// TIA Portal project "SortingLine_Project" (V18)

(* hardware
DEVICE "S7-1200 station_1"  S7-1200 Station
   slot 0: "Rack_0"  S7-1200 Rack  Rack  V1.0
   slot 1: "PLC_Sorting"  CPU 1214C DC/DC/DC  6ES7 214-1AG40-0XB0  V4.6
*)

// ===== PLC "PLC_Sorting"  CPU 1214C DC/DC/DC =====

VAR_GLOBAL   // PLC tag table "Factory_IO_Outputs"
   "Q_Counter" AT %QD30 : DInt;   // Digital totalizer display unit located on the operator panel.
   "Q_EntryConveyor" AT %Q0.1 : Bool;   // Drives the second section of the entry lane towards the turntable.
   "Q_FeederConveyor" AT %Q0.0 : Bool;   // Drives the first entry section right beneath the box emitter.
   "Q_GreenIndicator" AT %Q0.7 : Bool;   // Constant green indicates system is running active cycles.
   "Q_LeftConveyor" AT %Q0.5 : Bool;   // Drives the left clearance exit lane.
   "Q_Load" AT %Q0.2 : Bool;   // Runs internal turntable rollers forward to pull a box inside.
   "Q_RedIndicator" AT %Q1.1 : Bool;   // Constant red indicates system is idle/stopped.
   "Q_ResetLight" AT %Q1.3 : Bool;   // Active when safety is tripped and waiting for Reset.
   "Q_RightConveyor" AT %Q0.6 : Bool;   // Drives the right clearance exit lane.
   "Q_StartLight" AT %Q1.2 : Bool;   // Follows the Run state.
   "Q_StopLight" AT %Q1.4 : Bool;   // Active when cycle is offline.
   "Q_Turn" AT %Q0.4 : Bool;   // Swivels the turntable mechanism 90° clockwise.
   "Q_Unload" AT %Q0.3 : Bool;   // Runs internal turntable rollers backward to eject a box out to the left lane.
   "Q_YellowIndicator" AT %Q1.0 : Bool;   // Active on safety Fault or when system is in Manual mode.
   "Q_RemoverLeft" AT %Q1.5 : Bool;   // Instantly deletes boxes at the left exit limit.
   "Q_RemoverRight" AT %Q1.6 : Bool;   // Instantly deletes boxes at the right exit limit.
   "Q_Emit" AT %Q1.7 : Bool;   // Continuous TRUE spawns boxes sequentially.
END_VAR

VAR_GLOBAL   // PLC tag table "Factory_IO_Inputs"
   "I_atBack" AT %I2.1 : Bool;   // Confirms a box has fully cleared the entry area.
   "I_atEntry" AT %I0.0 : Bool;   // Detects box emergence.
   "I_atFront" AT %I0.6 : Bool;   // Prevents part collisions.
   "I_atLeftEntry" AT %I1.0 : Bool;   // Confirms the box has successfully transitioned onto the Left exit conveyor.
   "I_atLeftExit" AT %I1.2 : Bool;   // Drops to FALSE when a box reaches the left remover.
   "I_atLoadPosition" AT %I0.4 : Bool;   // TRUE when turntable is at 0° (aligned with entry).
   "I_atRightEntry" AT %I0.7 : Bool;   // Confirms the box has successfully transitioned onto the Right exit conveyor.
   "I_atRightExit" AT %I1.1 : Bool;   // Drops to FALSE when a box reaches the right remover.
   "I_atTurntableEntry" AT %I0.3 : Bool;   // Center reflective sensor inside the turntable. Used for precise stopping.
   "I_atUnloadPosition" AT %I0.5 : Bool;   // TRUE when turntable has completed its 90° clockwise rotation.
   "I_Auto" AT %I1.7 : Bool;   // Selector in Auto position.
   "I_Manual" AT %I2.2 : Bool;   // Selector in Manual position.
   "I_EmergencyStop" AT %I1.6 : Bool;   // TRUE when healthy, drops to FALSE when pressed.
   "I_LowBox" AT %I0.1 : Bool;   // Active (TRUE) for both low and high boxes.
   "I_Reset" AT %I1.4 : Bool;   // Clears safety fault latches.
   "I_Start" AT %I1.3 : Bool;   // Triggers the cycle run latch.
   "I_Stop" AT %I1.5 : Bool;   // TRUE at rest, drops to FALSE to request a cycle stop.
   "I_HighBox" AT %I0.2 : Bool;   // Active (TRUE) only alongside LowBox for high boxes.
END_VAR

TYPE "UDT_ActuatorCmd"
   STRUCT
      EntryConveyor : Bool;
      FeederConveyor : Bool;
      LeftConveyor : Bool;
      RightConveyor : Bool;
      Load : Bool;
      Unload : Bool;
      Turn : Bool;
      Emit : Bool;
      RemoverLeft : Bool := true;
      RemoverRight : Bool := true;
   END_STRUCT;
END_TYPE

DATA_BLOCK "DB_Machine"   // DB1
TITLE = Global Machine Status and Shared Data Registers
{ S7_Optimized_Access := 'TRUE' }
AUTHOR : HoraEmbedded
VERSION : 0.1
// Global Data Block (DB) serving as the main internal memory exchange registry for the system. Contains structured variables for system operating flags (Run, Fault, Modes), active part counters (Total, Left, Right), manual control parameters generated by the operator panel, and live engineering settings such as the box centering delay time variable.
   VAR
      Run : Bool;
      Fault : Bool;
      StopPending : Bool;
      AutoMode : Bool;
      ManualMode : Bool;
      CycleIdle : Bool;
      CountLeft : DInt;
      CountRight : DInt;
      CountTotal : DInt;
      AutoCmd : "UDT_ActuatorCmd";
      ManCmd : "UDT_ActuatorCmd";
      SortStep : DInt;
      ExitIdleHigh : Bool;
      ClearCounters : Bool;
      CenterTime : Time := T#2s;
   END_VAR
BEGIN
END_DATA_BLOCK

DATA_BLOCK "FB_ModeManager_DB"   // DB2
{ S7_Optimized_Access := 'TRUE' }
VERSION : 0.1
// stored: InstanceOfName FB_ModeManager
"FB_ModeManager"
BEGIN
END_DATA_BLOCK

DATA_BLOCK "FB_SortingLogic_DB"   // DB3
{ S7_Optimized_Access := 'TRUE' }
VERSION : 0.1
// stored: InstanceOfName FB_SortingLogic
"FB_SortingLogic"
BEGIN
END_DATA_BLOCK

FUNCTION_BLOCK "FB_ModeManager"   // FB1, LAD
TITLE = Machine Modes and Safety Interlocking Manager
{ S7_Optimized_Access := 'TRUE' }
AUTHOR : HoraEmbedded
VERSION : 0.1
// Monitors physical safety devices and panel inputs to manage operational states. Implements Normally Closed (NC) healthy monitoring for the Emergency Stop button, manages the manual safety fault latch (SR flip-flop), and handles the cycle stop requests (StopPending logic). It ensures a clean segregation between AutoMode and ManualMode to prevent overlapping operational commands.
   VAR_INPUT
      i_Start : Bool;   // Start pushbutton
      i_StopNC : Bool;   // Stop pushbutton
      i_EstopNC : Bool;   // Emergency stop
      i_Reset : Bool;   // Reset pushbutton
      i_Auto : Bool;   // Selector in Auto
      i_Manual : Bool;   // Selector in Manual
      i_CycleIdle : Bool;   // No box being processed
   END_VAR
   VAR_OUTPUT
      o_Run : Bool;
      o_Fault : Bool;
      o_StopPending : Bool;
      o_AutoMode : Bool;
      o_ManualMode : Bool;
   END_VAR
   VAR
      s_EdgeStart : Bool;   // Edge memory bits
      s_EdgeReset : Bool;   // Edge memory bits
   END_VAR
   VAR_TEMP
      t_StartPulse : Bool;   // One scan pulses
      t_ResetPulse : Bool;   // One scan pulses
   END_VAR
   VAR_TEMP   // added for the SCL form of the ladder/FBD networks
      _w1 : Bool;
   END_VAR
BEGIN

REGION Network 1: Auto mode
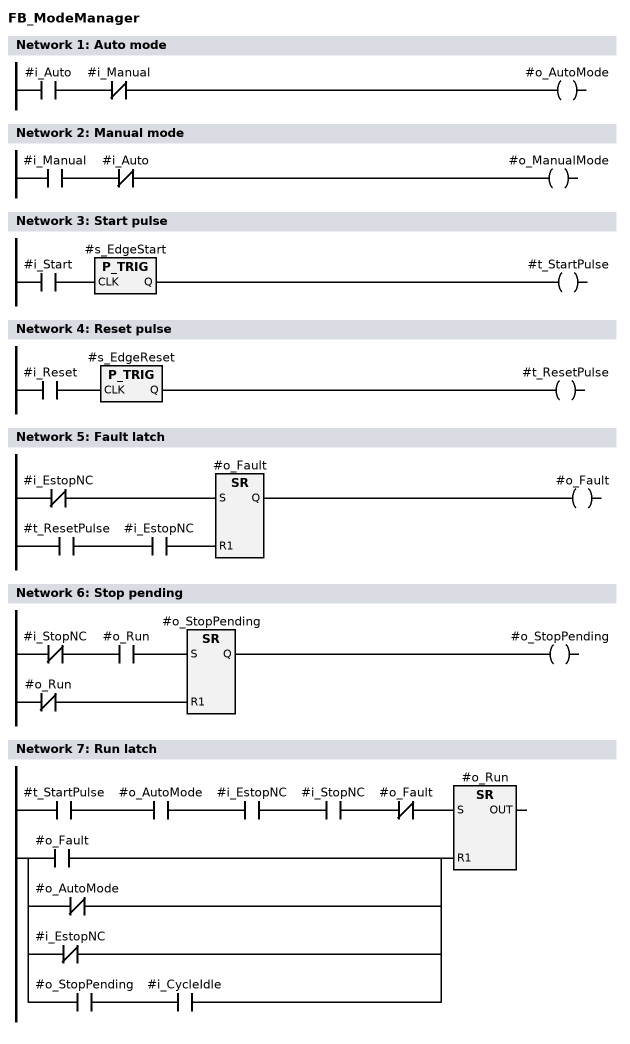
   RUNG wire#powerrail
      Contact( #i_Auto )
      I_Contact( #i_Manual )
      Coil( #o_AutoMode )
   END_RUNG
   // the same network as SCL:
   #o_AutoMode := #i_Auto AND NOT #i_Manual;
END_REGION

REGION Network 2: Manual mode
   RUNG wire#powerrail
      Contact( #i_Manual )
      I_Contact( #i_Auto )
      Coil( #o_ManualMode )
   END_RUNG
   // the same network as SCL:
   #o_ManualMode := #i_Manual AND NOT #i_Auto;
END_REGION

REGION Network 3: Start pulse
   RUNG wire#powerrail
      Contact( #i_Start )
      P_Trig( #s_EdgeStart )
      Coil( #t_StartPulse )
   END_RUNG
   // the same network as SCL:
   #_w1 := #i_Start AND NOT #s_EdgeStart;   // rising edge
   #s_EdgeStart := #i_Start;
   #t_StartPulse := #_w1;
END_REGION

REGION Network 4: Reset pulse
   RUNG wire#powerrail
      Contact( #i_Reset )
      P_Trig( #s_EdgeReset )
      Coil( #t_ResetPulse )
   END_RUNG
   // the same network as SCL:
   #_w1 := #i_Reset AND NOT #s_EdgeReset;   // rising edge
   #s_EdgeReset := #i_Reset;
   #t_ResetPulse := #_w1;
END_REGION

REGION Network 5: Fault latch
   RUNG wire#powerrail
      I_Contact( #i_EstopNC )
      S_SR(operand := #o_Fault, r1 := wire#w1)
      Coil( #o_Fault )
   END_RUNG
   RUNG wire#powerrail
      Contact( #t_ResetPulse )
      Contact( #i_EstopNC )
   END_RUNG wire#w1
   // the same network as SCL:
   IF NOT #i_EstopNC THEN
       #o_Fault := TRUE;   // SR flip-flop
   END_IF;
   IF #t_ResetPulse AND #i_EstopNC THEN #o_Fault := FALSE; END_IF;
   #o_Fault := #o_Fault;
END_REGION

REGION Network 6: Stop pending
   RUNG wire#powerrail
      I_Contact( #i_StopNC )
      Contact( #o_Run )
      S_SR(operand := #o_StopPending, r1 := wire#w1)
      Coil( #o_StopPending )
   END_RUNG
   RUNG wire#powerrail
      I_Contact( #o_Run )
   END_RUNG wire#w1
   // the same network as SCL:
   IF NOT #i_StopNC AND #o_Run THEN
       #o_StopPending := TRUE;   // SR flip-flop
   END_IF;
   IF NOT #o_Run THEN #o_StopPending := FALSE; END_IF;
   #o_StopPending := #o_StopPending;
END_REGION

REGION Network 7: Run latch
   RUNG wire#powerrail
      Contact( #t_StartPulse )
      Contact( #o_AutoMode )
      Contact( #i_EstopNC )
      Contact( #i_StopNC )
      I_Contact( #o_Fault )
      S_SR(operand := #o_Run, r1 := wire#w1)
   END_RUNG
   RUNG wire#powerrail
      Contact( #o_Fault )
   END_RUNG wire#w1
   RUNG wire#powerrail
      I_Contact( #o_AutoMode )
   END_RUNG wire#w1
   RUNG wire#powerrail
      I_Contact( #i_EstopNC )
   END_RUNG wire#w1
   RUNG wire#powerrail
      Contact( #o_StopPending )
      Contact( #i_CycleIdle )
   END_RUNG wire#w1
   // the same network as SCL:
   IF #t_StartPulse AND #o_AutoMode AND #i_EstopNC AND #i_StopNC AND NOT #o_Fault THEN
       #o_Run := TRUE;   // SR flip-flop
   END_IF;
   IF #o_Fault OR NOT #o_AutoMode OR NOT #i_EstopNC OR (#o_StopPending AND #i_CycleIdle) THEN
       #o_Run := FALSE;
   END_IF;
END_REGION
END_FUNCTION_BLOCK

FUNCTION_BLOCK "FB_SortingLogic"   // FB2, LAD
TITLE = Pipelined Box Sorting Sequence (State Machine)
{ S7_Optimized_Access := 'TRUE' }
AUTHOR : HoraEmbedded
VERSION : 0.1
// Implements the continuous automatic sorting sequence using a customized sequential state machine (Steps 0 to 5). Manages entry box generation, calculates sensor filtration via an independent centering timer block, tracks multiple parts in transit using dedicated software registers (In-Transit counters), and automatically routes boxes based on height measurements recorded by the light curtain.
   VAR_INPUT
      i_Run : Bool;
      i_StopPending : Bool;
      i_ClearCounters : Bool;
      i_ExitIdleHigh : Bool;
      i_atEntry : Bool;
      i_atLoadPosition : Bool;
      i_atTurntableEntry : Bool;
      i_atUnloadPosition : Bool;
      i_HighBox : Bool;
      i_atLeftEntry : Bool;
      i_atRightEntry : Bool;
      i_atLeftExit : Bool;
      i_atRightExit : Bool;
      i_CenterTime : Time;
      i_atFront : Bool;
   END_VAR
   VAR_OUTPUT
      o_CycleIdle : Bool;
      o_Step : DInt;
   END_VAR
   VAR_IN_OUT
      io_Cmd : "UDT_ActuatorCmd";
      io_CountLeft : DInt;
      io_CountRight : DInt;
      io_CountTotal : DInt;
   END_VAR
   VAR
      s_Step : DInt;
      s_SeenHigh : Bool;
      s_EdgeExitLeft : Bool;
      s_EdgeExitRight : Bool;
      s_TonEmit : IEC_TIMER;
      s_TonCenter : IEC_TIMER;
      s_atEntrySeen : Bool;
      s_LeftInTransit : DInt;
      s_RightInTransit : DInt;
      s_EdgeLeftEntry : Bool;
      s_EdgeRightEntry : Bool;
   END_VAR
   VAR_TEMP
      t_ExitLeftActive : Bool;
      t_ExitRightActive : Bool;
      t_ExitLeftPulse : Bool;
      t_ExitRightPulse : Bool;
      t_ChosenEntry : Bool;
      t_LeftEntryPulse : Bool;
      t_RightEntryPulse : Bool;
   END_VAR
   VAR_TEMP   // added for the SCL form of the ladder/FBD networks
      _w1 : Bool;
   END_VAR
BEGIN

REGION Network 1: exit left active
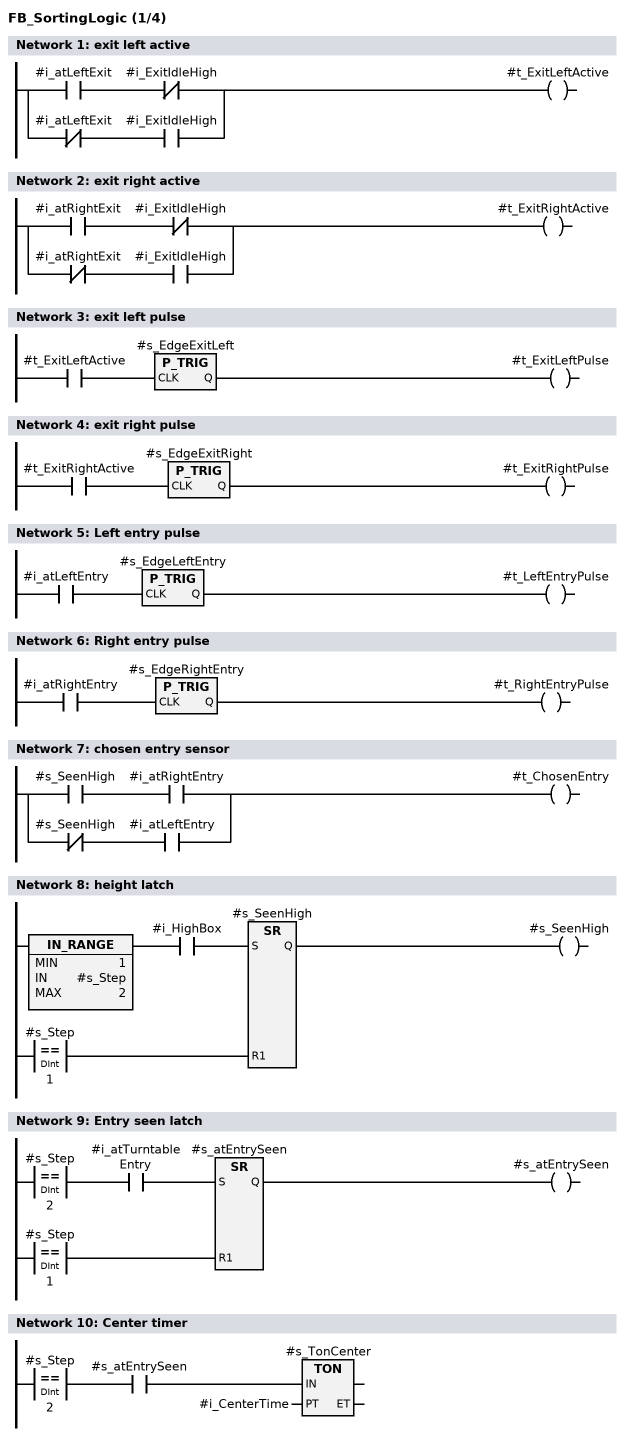
   RUNG wire#powerrail
      Contact( #i_atLeftExit )
      I_Contact( #i_ExitIdleHigh )
      wire#w1
      Coil( #t_ExitLeftActive )
   END_RUNG
   RUNG wire#powerrail
      I_Contact( #i_atLeftExit )
      Contact( #i_ExitIdleHigh )
   END_RUNG wire#w1
   // the same network as SCL:
   #t_ExitLeftActive := (#i_atLeftExit AND NOT #i_ExitIdleHigh) OR (NOT #i_atLeftExit AND #i_ExitIdleHigh);
END_REGION

REGION Network 2: exit right active
   RUNG wire#powerrail
      Contact( #i_atRightExit )
      I_Contact( #i_ExitIdleHigh )
      wire#w1
      Coil( #t_ExitRightActive )
   END_RUNG
   RUNG wire#powerrail
      I_Contact( #i_atRightExit )
      Contact( #i_ExitIdleHigh )
   END_RUNG wire#w1
   // the same network as SCL:
   #t_ExitRightActive := (#i_atRightExit AND NOT #i_ExitIdleHigh) OR (NOT #i_atRightExit AND #i_ExitIdleHigh);
END_REGION

REGION Network 3: exit left pulse
   RUNG wire#powerrail
      Contact( #t_ExitLeftActive )
      P_Trig( #s_EdgeExitLeft )
      Coil( #t_ExitLeftPulse )
   END_RUNG
   // the same network as SCL:
   #_w1 := #t_ExitLeftActive AND NOT #s_EdgeExitLeft;   // rising edge
   #s_EdgeExitLeft := #t_ExitLeftActive;
   #t_ExitLeftPulse := #_w1;
END_REGION

REGION Network 4: exit right pulse
   RUNG wire#powerrail
      Contact( #t_ExitRightActive )
      P_Trig( #s_EdgeExitRight )
      Coil( #t_ExitRightPulse )
   END_RUNG
   // the same network as SCL:
   #_w1 := #t_ExitRightActive AND NOT #s_EdgeExitRight;   // rising edge
   #s_EdgeExitRight := #t_ExitRightActive;
   #t_ExitRightPulse := #_w1;
END_REGION

REGION Network 5: Left entry pulse
   RUNG wire#powerrail
      Contact( #i_atLeftEntry )
      P_Trig( #s_EdgeLeftEntry )
      Coil( #t_LeftEntryPulse )
   END_RUNG
   // the same network as SCL:
   #_w1 := #i_atLeftEntry AND NOT #s_EdgeLeftEntry;   // rising edge
   #s_EdgeLeftEntry := #i_atLeftEntry;
   #t_LeftEntryPulse := #_w1;
END_REGION

REGION Network 6: Right entry pulse
   RUNG wire#powerrail
      Contact( #i_atRightEntry )
      P_Trig( #s_EdgeRightEntry )
      Coil( #t_RightEntryPulse )
   END_RUNG
   // the same network as SCL:
   #_w1 := #i_atRightEntry AND NOT #s_EdgeRightEntry;   // rising edge
   #s_EdgeRightEntry := #i_atRightEntry;
   #t_RightEntryPulse := #_w1;
END_REGION

REGION Network 7: chosen entry sensor
   RUNG wire#powerrail
      Contact( #s_SeenHigh )
      Contact( #i_atRightEntry )
      wire#w1
      Coil( #t_ChosenEntry )
   END_RUNG
   RUNG wire#powerrail
      I_Contact( #s_SeenHigh )
      Contact( #i_atLeftEntry )
   END_RUNG wire#w1
   // the same network as SCL:
   #t_ChosenEntry := (#s_SeenHigh AND #i_atRightEntry) OR (NOT #s_SeenHigh AND #i_atLeftEntry);
END_REGION

REGION Network 8: height latch
   RUNG wire#powerrail
      { S7_Templates := "SrcType := DInt" } InRange(min := 1, in := #s_Step, max := 2)
      Contact( #i_HighBox )
      S_SR(operand := #s_SeenHigh, r1 := wire#w1)
      Coil( #s_SeenHigh )
   END_RUNG
   RUNG wire#powerrail
      { S7_Templates := "SrcType := DInt" } EQ_Contact(in1 := #s_Step, in2 := 1)
   END_RUNG wire#w1
   // the same network as SCL:
   IF (1 <= #s_Step) AND (#s_Step <= 2) AND #i_HighBox THEN
       #s_SeenHigh := TRUE;   // SR flip-flop
   END_IF;
   IF #s_Step = 1 THEN #s_SeenHigh := FALSE; END_IF;
   #s_SeenHigh := #s_SeenHigh;
END_REGION

REGION Network 9: Entry seen latch
   RUNG wire#powerrail
      { S7_Templates := "SrcType := DInt" } EQ_Contact(in1 := #s_Step, in2 := 2)
      Contact( #i_atTurntableEntry )
      S_SR(operand := #s_atEntrySeen, r1 := wire#w1)
      Coil( #s_atEntrySeen )
   END_RUNG
   RUNG wire#powerrail
      { S7_Templates := "SrcType := DInt" } EQ_Contact(in1 := #s_Step, in2 := 1)
   END_RUNG wire#w1
   // the same network as SCL:
   IF (#s_Step = 2) AND #i_atTurntableEntry THEN
       #s_atEntrySeen := TRUE;   // SR flip-flop
   END_IF;
   IF #s_Step = 1 THEN #s_atEntrySeen := FALSE; END_IF;
   #s_atEntrySeen := #s_atEntrySeen;
END_REGION

REGION Network 10: Center timer
   #s_TonCenter.TON(IN := (#s_Step = 2) AND #s_atEntrySeen, PT := #i_CenterTime);
END_REGION

REGION Network 11: T4 to 5 (#s_Step := 5)
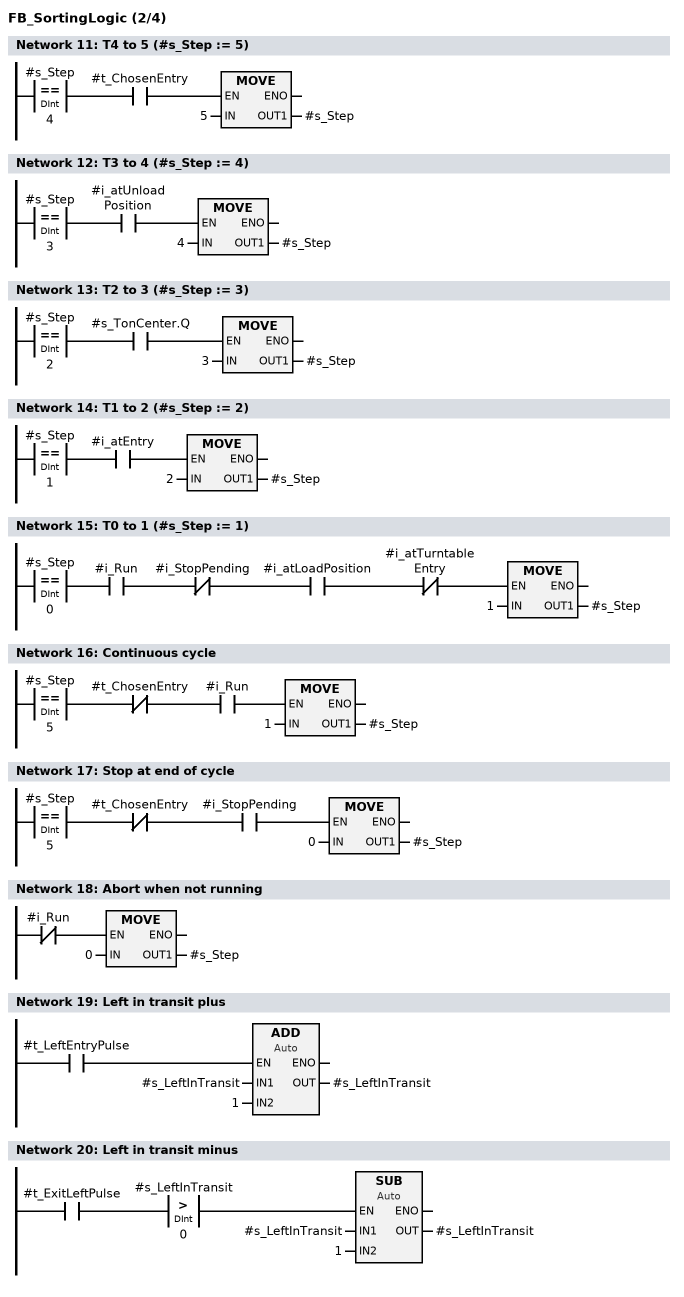
   RUNG wire#powerrail
      { S7_Templates := "SrcType := DInt" } EQ_Contact(in1 := #s_Step, in2 := 4)
      Contact( #t_ChosenEntry )
      Move(in := 5, out1 => #s_Step)
   END_RUNG
   // the same network as SCL:
   IF (#s_Step = 4) AND #t_ChosenEntry THEN #s_Step := 5; END_IF;
END_REGION

REGION Network 12: T3 to 4 (#s_Step := 4)
   RUNG wire#powerrail
      { S7_Templates := "SrcType := DInt" } EQ_Contact(in1 := #s_Step, in2 := 3)
      Contact( #i_atUnloadPosition )
      Move(in := 4, out1 => #s_Step)
   END_RUNG
   // the same network as SCL:
   IF (#s_Step = 3) AND #i_atUnloadPosition THEN #s_Step := 4; END_IF;
END_REGION

REGION Network 13: T2 to 3 (#s_Step := 3)
   RUNG wire#powerrail
      { S7_Templates := "SrcType := DInt" } EQ_Contact(in1 := #s_Step, in2 := 2)
      Contact( #s_TonCenter.Q )
      Move(in := 3, out1 => #s_Step)
   END_RUNG
   // the same network as SCL:
   IF (#s_Step = 2) AND #s_TonCenter.Q THEN #s_Step := 3; END_IF;
END_REGION

REGION Network 14: T1 to 2 (#s_Step := 2)
   RUNG wire#powerrail
      { S7_Templates := "SrcType := DInt" } EQ_Contact(in1 := #s_Step, in2 := 1)
      Contact( #i_atEntry )
      Move(in := 2, out1 => #s_Step)
   END_RUNG
   // the same network as SCL:
   IF (#s_Step = 1) AND #i_atEntry THEN #s_Step := 2; END_IF;
END_REGION

REGION Network 15: T0 to 1 (#s_Step := 1)
   RUNG wire#powerrail
      { S7_Templates := "SrcType := DInt" } EQ_Contact(in1 := #s_Step, in2 := 0)
      Contact( #i_Run )
      I_Contact( #i_StopPending )
      Contact( #i_atLoadPosition )
      I_Contact( #i_atTurntableEntry )
      Move(in := 1, out1 => #s_Step)
   END_RUNG
   // the same network as SCL:
   IF (#s_Step = 0) AND #i_Run AND NOT #i_StopPending AND #i_atLoadPosition AND NOT #i_atTurntableEntry THEN
       #s_Step := 1;
   END_IF;
END_REGION

REGION Network 16: Continuous cycle
   RUNG wire#powerrail
      { S7_Templates := "SrcType := DInt" } EQ_Contact(in1 := #s_Step, in2 := 5)
      I_Contact( #t_ChosenEntry )
      Contact( #i_Run )
      Move(in := 1, out1 => #s_Step)
   END_RUNG
   // the same network as SCL:
   IF (#s_Step = 5) AND NOT #t_ChosenEntry AND #i_Run THEN #s_Step := 1; END_IF;
END_REGION

REGION Network 17: Stop at end of cycle
   RUNG wire#powerrail
      { S7_Templates := "SrcType := DInt" } EQ_Contact(in1 := #s_Step, in2 := 5)
      I_Contact( #t_ChosenEntry )
      Contact( #i_StopPending )
      Move(in := 0, out1 => #s_Step)
   END_RUNG
   // the same network as SCL:
   IF (#s_Step = 5) AND NOT #t_ChosenEntry AND #i_StopPending THEN #s_Step := 0; END_IF;
END_REGION

REGION Network 18: Abort when not running
   RUNG wire#powerrail
      I_Contact( #i_Run )
      Move(in := 0, out1 => #s_Step)
   END_RUNG
   // the same network as SCL:
   IF NOT #i_Run THEN #s_Step := 0; END_IF;
END_REGION

REGION Network 19: Left in transit plus
   RUNG wire#powerrail
      Contact( #t_LeftEntryPulse )
      Add(in1 := #s_LeftInTransit, in2 := 1, out => #s_LeftInTransit)
   END_RUNG
   // the same network as SCL:
   IF #t_LeftEntryPulse THEN #s_LeftInTransit := #s_LeftInTransit + 1; END_IF;
END_REGION

REGION Network 20: Left in transit minus
   RUNG wire#powerrail
      Contact( #t_ExitLeftPulse )
      { S7_Templates := "SrcType := DInt" } GT_Contact(in1 := #s_LeftInTransit, in2 := 0)
      Sub(in1 := #s_LeftInTransit, in2 := 1, out => #s_LeftInTransit)
   END_RUNG
   // the same network as SCL:
   IF #t_ExitLeftPulse AND (#s_LeftInTransit > 0) THEN #s_LeftInTransit := #s_LeftInTransit - 1; END_IF;
END_REGION

REGION Network 21: Left in transit clear
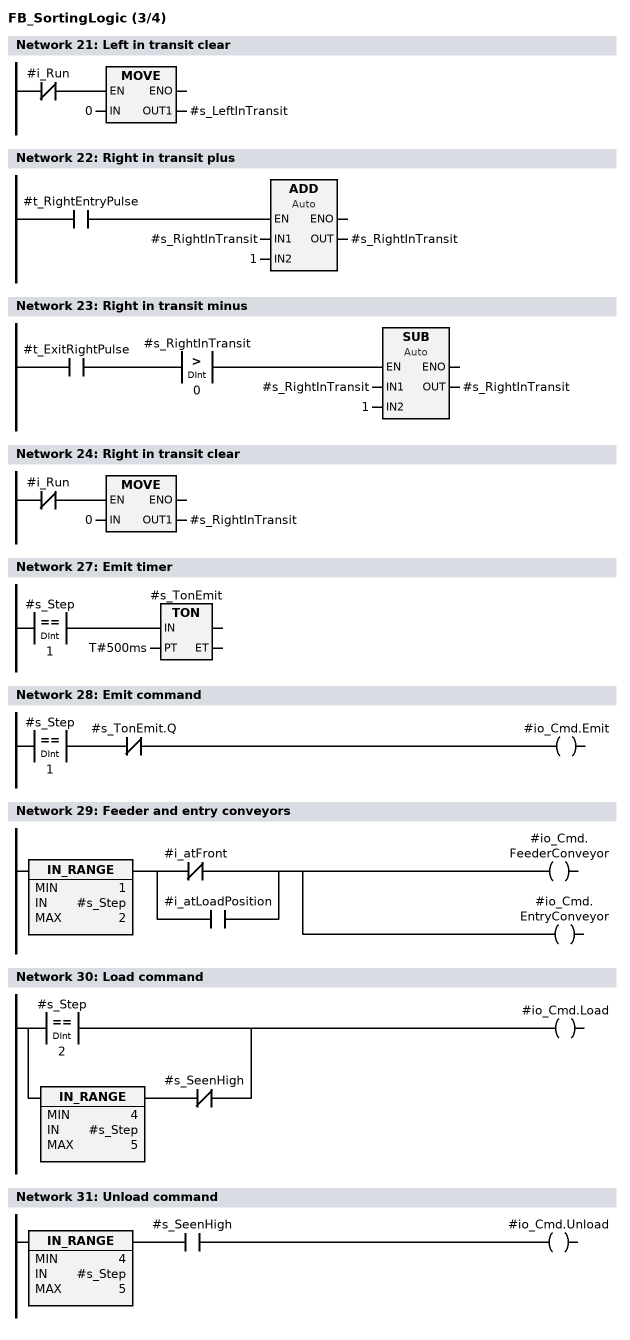
   RUNG wire#powerrail
      I_Contact( #i_Run )
      Move(in := 0, out1 => #s_LeftInTransit)
   END_RUNG
   // the same network as SCL:
   IF NOT #i_Run THEN #s_LeftInTransit := 0; END_IF;
END_REGION

REGION Network 22: Right in transit plus
   RUNG wire#powerrail
      Contact( #t_RightEntryPulse )
      Add(in1 := #s_RightInTransit, in2 := 1, out => #s_RightInTransit)
   END_RUNG
   // the same network as SCL:
   IF #t_RightEntryPulse THEN #s_RightInTransit := #s_RightInTransit + 1; END_IF;
END_REGION

REGION Network 23: Right in transit minus
   RUNG wire#powerrail
      Contact( #t_ExitRightPulse )
      { S7_Templates := "SrcType := DInt" } GT_Contact(in1 := #s_RightInTransit, in2 := 0)
      Sub(in1 := #s_RightInTransit, in2 := 1, out => #s_RightInTransit)
   END_RUNG
   // the same network as SCL:
   IF #t_ExitRightPulse AND (#s_RightInTransit > 0) THEN #s_RightInTransit := #s_RightInTransit - 1; END_IF;
END_REGION

REGION Network 24: Right in transit clear
   RUNG wire#powerrail
      I_Contact( #i_Run )
      Move(in := 0, out1 => #s_RightInTransit)
   END_RUNG
   // the same network as SCL:
   IF NOT #i_Run THEN #s_RightInTransit := 0; END_IF;
END_REGION

REGION Network 25: Continuous cycle
END_REGION

REGION Network 26: Stop at end of cycle
END_REGION

REGION Network 27: Emit timer
   #s_TonEmit.TON(IN := #s_Step = 1, PT := T#500ms);
END_REGION

REGION Network 28: Emit command
   RUNG wire#powerrail
      { S7_Templates := "SrcType := DInt" } EQ_Contact(in1 := #s_Step, in2 := 1)
      I_Contact( #s_TonEmit.Q )
      Coil( #io_Cmd.Emit )
   END_RUNG
   // the same network as SCL:
   #io_Cmd.Emit := (#s_Step = 1) AND NOT #s_TonEmit.Q;
END_REGION

REGION Network 29: Feeder and entry conveyors
   RUNG wire#powerrail
      { S7_Templates := "SrcType := DInt" } InRange(min := 1, in := #s_Step, max := 2)
      wire#w1
      I_Contact( #i_atFront )
      wire#w2
      Coil( #io_Cmd.FeederConveyor )
   END_RUNG
   RUNG wire#w1
      Contact( #i_atLoadPosition )
   END_RUNG wire#w2
   RUNG wire#w2
      Coil( #io_Cmd.EntryConveyor )
   END_RUNG
   // the same network as SCL:
   #io_Cmd.FeederConveyor := (1 <= #s_Step) AND (#s_Step <= 2) AND (NOT #i_atFront OR #i_atLoadPosition);
   #io_Cmd.EntryConveyor := #io_Cmd.FeederConveyor;
END_REGION

REGION Network 30: Load command
   RUNG wire#powerrail
      { S7_Templates := "SrcType := DInt" } EQ_Contact(in1 := #s_Step, in2 := 2)
      wire#w1
      Coil( #io_Cmd.Load )
   END_RUNG
   RUNG wire#powerrail
      { S7_Templates := "SrcType := DInt" } InRange(min := 4, in := #s_Step, max := 5)
      I_Contact( #s_SeenHigh )
   END_RUNG wire#w1
   // the same network as SCL:
   #io_Cmd.Load := (#s_Step = 2) OR ((4 <= #s_Step) AND (#s_Step <= 5) AND NOT #s_SeenHigh);
END_REGION

REGION Network 31: Unload command
   RUNG wire#powerrail
      { S7_Templates := "SrcType := DInt" } InRange(min := 4, in := #s_Step, max := 5)
      Contact( #s_SeenHigh )
      Coil( #io_Cmd.Unload )
   END_RUNG
   // the same network as SCL:
   #io_Cmd.Unload := (4 <= #s_Step) AND (#s_Step <= 5) AND #s_SeenHigh;
END_REGION

REGION Network 32: Turn command
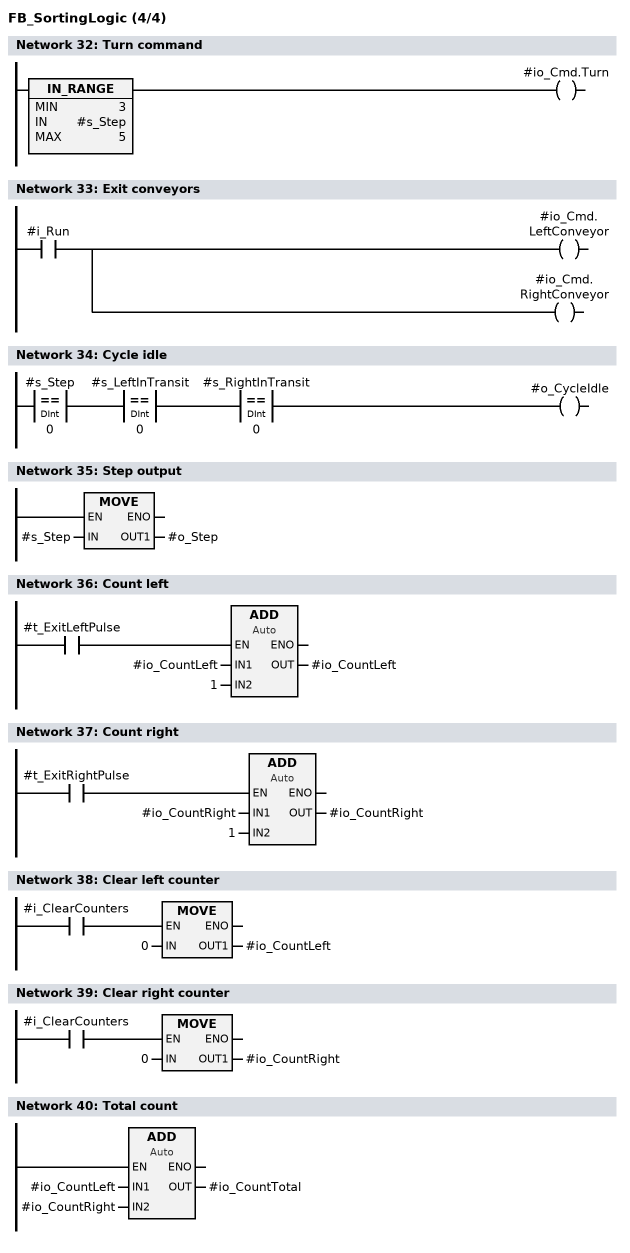
   RUNG wire#powerrail
      { S7_Templates := "SrcType := DInt" } InRange(min := 3, in := #s_Step, max := 5)
      Coil( #io_Cmd.Turn )
   END_RUNG
   // the same network as SCL:
   #io_Cmd.Turn := (3 <= #s_Step) AND (#s_Step <= 5);
END_REGION

REGION Network 33: Exit conveyors
   RUNG wire#powerrail
      Contact( #i_Run )
      wire#w1
      Coil( #io_Cmd.LeftConveyor )
   END_RUNG
   RUNG wire#w1
      Coil( #io_Cmd.RightConveyor )
   END_RUNG
   // the same network as SCL:
   #io_Cmd.LeftConveyor := #i_Run;
   #io_Cmd.RightConveyor := #i_Run;
END_REGION

REGION Network 34: Cycle idle
   RUNG wire#powerrail
      { S7_Templates := "SrcType := DInt" } EQ_Contact(in1 := #s_Step, in2 := 0)
      { S7_Templates := "SrcType := DInt" } EQ_Contact(in1 := #s_LeftInTransit, in2 := 0)
      { S7_Templates := "SrcType := DInt" } EQ_Contact(in1 := #s_RightInTransit, in2 := 0)
      Coil( #o_CycleIdle )
   END_RUNG
   // the same network as SCL:
   #o_CycleIdle := (#s_Step = 0) AND (#s_LeftInTransit = 0) AND (#s_RightInTransit = 0);
END_REGION

REGION Network 35: Step output
   RUNG wire#powerrail
      Move(in := #s_Step, out1 => #o_Step)
   END_RUNG
   // the same network as SCL:
   #o_Step := #s_Step;
END_REGION

REGION Network 36: Count left
   RUNG wire#powerrail
      Contact( #t_ExitLeftPulse )
      Add(in1 := #io_CountLeft, in2 := 1, out => #io_CountLeft)
   END_RUNG
   // the same network as SCL:
   IF #t_ExitLeftPulse THEN #io_CountLeft := #io_CountLeft + 1; END_IF;
END_REGION

REGION Network 37: Count right
   RUNG wire#powerrail
      Contact( #t_ExitRightPulse )
      Add(in1 := #io_CountRight, in2 := 1, out => #io_CountRight)
   END_RUNG
   // the same network as SCL:
   IF #t_ExitRightPulse THEN #io_CountRight := #io_CountRight + 1; END_IF;
END_REGION

REGION Network 38: Clear left counter
   RUNG wire#powerrail
      Contact( #i_ClearCounters )
      Move(in := 0, out1 => #io_CountLeft)
   END_RUNG
   // the same network as SCL:
   IF #i_ClearCounters THEN #io_CountLeft := 0; END_IF;
END_REGION

REGION Network 39: Clear right counter
   RUNG wire#powerrail
      Contact( #i_ClearCounters )
      Move(in := 0, out1 => #io_CountRight)
   END_RUNG
   // the same network as SCL:
   IF #i_ClearCounters THEN #io_CountRight := 0; END_IF;
END_REGION

REGION Network 40: Total count
   RUNG wire#powerrail
      Add(in1 := #io_CountLeft, in2 := #io_CountRight, out => #io_CountTotal)
   END_RUNG
   // the same network as SCL:
   #io_CountTotal := #io_CountLeft + #io_CountRight;
END_REGION
END_FUNCTION_BLOCK

FUNCTION "FC_outputs" : Void   // FC1, LAD
TITLE = Centralized Output Gating and Hardware Interlocks
{ S7_Optimized_Access := 'TRUE' }
AUTHOR : HoraEmbedded
VERSION : 0.1
// Serves as the single source of truth for all physical digital and analog outputs directed to the Factory I/O simulation panel. It gathers automatic commands generated by the state machine and manual commands from the watch table. It applies strict hardware safety interlocks (System Enable bit derived from the Emergency Stop state) before forcing any physical coil to prevent duplicate assignment conflicts.
   VAR_TEMP
      t_Enable : Bool;
   END_VAR
BEGIN

REGION Network 1: Enable
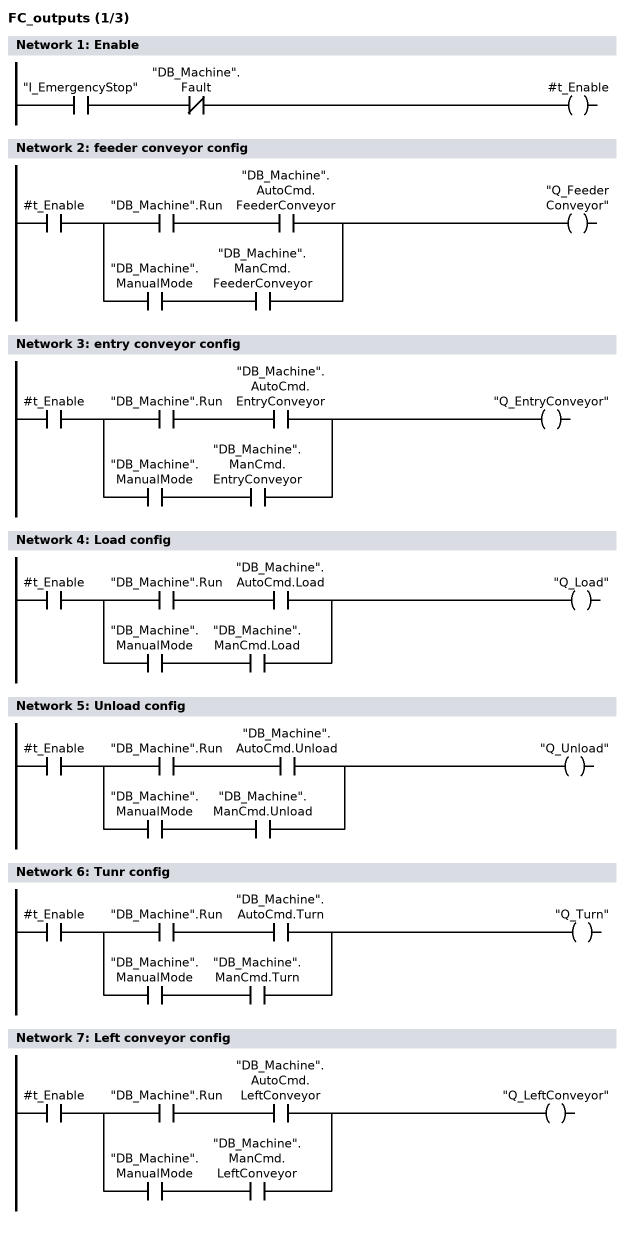
   RUNG wire#powerrail
      Contact( "I_EmergencyStop" )
      I_Contact( "DB_Machine".Fault )
      Coil( #t_Enable )
   END_RUNG
   // the same network as SCL:
   #t_Enable := "I_EmergencyStop" AND NOT "DB_Machine".Fault;
END_REGION

REGION Network 2: feeder conveyor config
   RUNG wire#powerrail
      Contact( #t_Enable )
      wire#w1
      Contact( "DB_Machine".Run )
      Contact( "DB_Machine".AutoCmd.FeederConveyor )
      wire#w2
      Coil( "Q_FeederConveyor" )
   END_RUNG
   RUNG wire#w1
      Contact( "DB_Machine".ManualMode )
      Contact( "DB_Machine".ManCmd.FeederConveyor )
   END_RUNG wire#w2
   // the same network as SCL:
   "Q_FeederConveyor" := #t_Enable AND (("DB_Machine".Run AND "DB_Machine".AutoCmd.FeederConveyor) OR ("DB_Machine".ManualMode AND "DB_Machine".ManCmd.FeederConveyor));
END_REGION

REGION Network 3: entry conveyor config
   RUNG wire#powerrail
      Contact( #t_Enable )
      wire#w1
      Contact( "DB_Machine".Run )
      Contact( "DB_Machine".AutoCmd.EntryConveyor )
      wire#w2
      Coil( "Q_EntryConveyor" )
   END_RUNG
   RUNG wire#w1
      Contact( "DB_Machine".ManualMode )
      Contact( "DB_Machine".ManCmd.EntryConveyor )
   END_RUNG wire#w2
   // the same network as SCL:
   "Q_EntryConveyor" := #t_Enable AND (("DB_Machine".Run AND "DB_Machine".AutoCmd.EntryConveyor) OR ("DB_Machine".ManualMode AND "DB_Machine".ManCmd.EntryConveyor));
END_REGION

REGION Network 4: Load config
   RUNG wire#powerrail
      Contact( #t_Enable )
      wire#w1
      Contact( "DB_Machine".Run )
      Contact( "DB_Machine".AutoCmd.Load )
      wire#w2
      Coil( "Q_Load" )
   END_RUNG
   RUNG wire#w1
      Contact( "DB_Machine".ManualMode )
      Contact( "DB_Machine".ManCmd.Load )
   END_RUNG wire#w2
   // the same network as SCL:
   "Q_Load" := #t_Enable AND (("DB_Machine".Run AND "DB_Machine".AutoCmd.Load) OR ("DB_Machine".ManualMode AND "DB_Machine".ManCmd.Load));
END_REGION

REGION Network 5: Unload config
   RUNG wire#powerrail
      Contact( #t_Enable )
      wire#w1
      Contact( "DB_Machine".Run )
      Contact( "DB_Machine".AutoCmd.Unload )
      wire#w2
      Coil( "Q_Unload" )
   END_RUNG
   RUNG wire#w1
      Contact( "DB_Machine".ManualMode )
      Contact( "DB_Machine".ManCmd.Unload )
   END_RUNG wire#w2
   // the same network as SCL:
   "Q_Unload" := #t_Enable AND (("DB_Machine".Run AND "DB_Machine".AutoCmd.Unload) OR ("DB_Machine".ManualMode AND "DB_Machine".ManCmd.Unload));
END_REGION

REGION Network 6: Tunr config
   RUNG wire#powerrail
      Contact( #t_Enable )
      wire#w1
      Contact( "DB_Machine".Run )
      Contact( "DB_Machine".AutoCmd.Turn )
      wire#w2
      Coil( "Q_Turn" )
   END_RUNG
   RUNG wire#w1
      Contact( "DB_Machine".ManualMode )
      Contact( "DB_Machine".ManCmd.Turn )
   END_RUNG wire#w2
   // the same network as SCL:
   "Q_Turn" := #t_Enable AND (("DB_Machine".Run AND "DB_Machine".AutoCmd.Turn) OR ("DB_Machine".ManualMode AND "DB_Machine".ManCmd.Turn));
END_REGION

REGION Network 7: Left conveyor config
   RUNG wire#powerrail
      Contact( #t_Enable )
      wire#w1
      Contact( "DB_Machine".Run )
      Contact( "DB_Machine".AutoCmd.LeftConveyor )
      wire#w2
      Coil( "Q_LeftConveyor" )
   END_RUNG
   RUNG wire#w1
      Contact( "DB_Machine".ManualMode )
      Contact( "DB_Machine".ManCmd.LeftConveyor )
   END_RUNG wire#w2
   // the same network as SCL:
   "Q_LeftConveyor" := #t_Enable AND (("DB_Machine".Run AND "DB_Machine".AutoCmd.LeftConveyor) OR ("DB_Machine".ManualMode AND "DB_Machine".ManCmd.LeftConveyor));
END_REGION

REGION Network 8: Right conveyor config
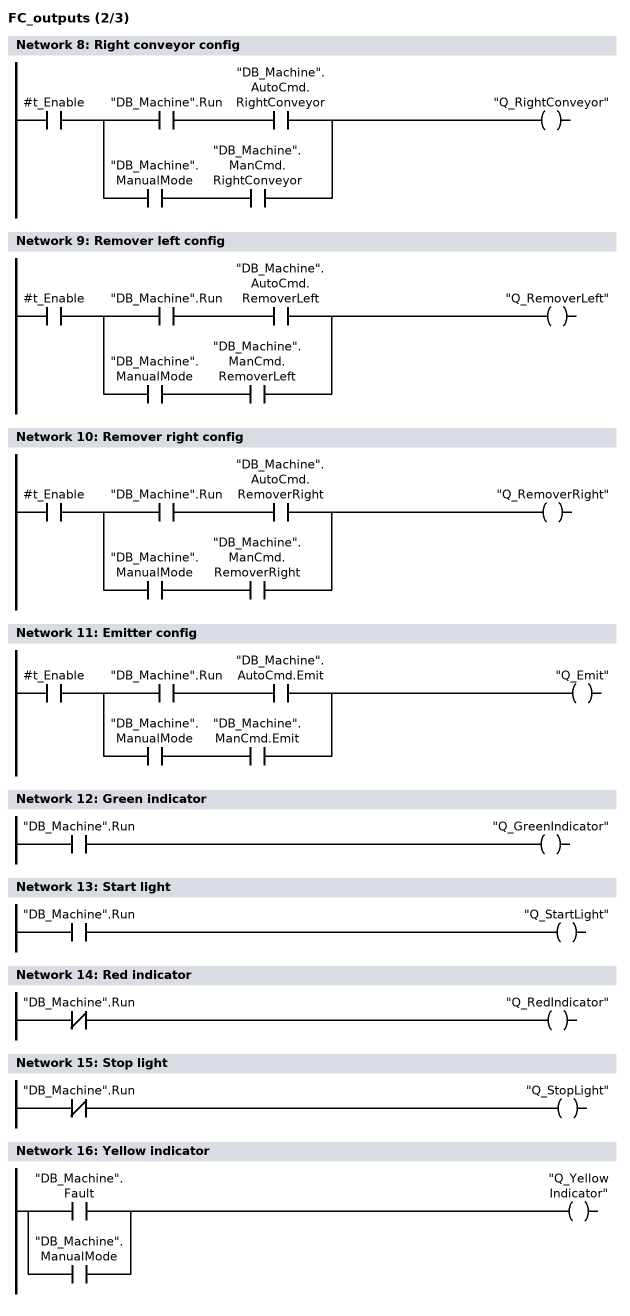
   RUNG wire#powerrail
      Contact( #t_Enable )
      wire#w1
      Contact( "DB_Machine".Run )
      Contact( "DB_Machine".AutoCmd.RightConveyor )
      wire#w2
      Coil( "Q_RightConveyor" )
   END_RUNG
   RUNG wire#w1
      Contact( "DB_Machine".ManualMode )
      Contact( "DB_Machine".ManCmd.RightConveyor )
   END_RUNG wire#w2
   // the same network as SCL:
   "Q_RightConveyor" := #t_Enable AND (("DB_Machine".Run AND "DB_Machine".AutoCmd.RightConveyor) OR ("DB_Machine".ManualMode AND "DB_Machine".ManCmd.RightConveyor));
END_REGION

REGION Network 9: Remover left config
   RUNG wire#powerrail
      Contact( #t_Enable )
      wire#w1
      Contact( "DB_Machine".Run )
      Contact( "DB_Machine".AutoCmd.RemoverLeft )
      wire#w2
      Coil( "Q_RemoverLeft" )
   END_RUNG
   RUNG wire#w1
      Contact( "DB_Machine".ManualMode )
      Contact( "DB_Machine".ManCmd.RemoverLeft )
   END_RUNG wire#w2
   // the same network as SCL:
   "Q_RemoverLeft" := #t_Enable AND (("DB_Machine".Run AND "DB_Machine".AutoCmd.RemoverLeft) OR ("DB_Machine".ManualMode AND "DB_Machine".ManCmd.RemoverLeft));
END_REGION

REGION Network 10: Remover right config
   RUNG wire#powerrail
      Contact( #t_Enable )
      wire#w1
      Contact( "DB_Machine".Run )
      Contact( "DB_Machine".AutoCmd.RemoverRight )
      wire#w2
      Coil( "Q_RemoverRight" )
   END_RUNG
   RUNG wire#w1
      Contact( "DB_Machine".ManualMode )
      Contact( "DB_Machine".ManCmd.RemoverRight )
   END_RUNG wire#w2
   // the same network as SCL:
   "Q_RemoverRight" := #t_Enable AND (("DB_Machine".Run AND "DB_Machine".AutoCmd.RemoverRight) OR ("DB_Machine".ManualMode AND "DB_Machine".ManCmd.RemoverRight));
END_REGION

REGION Network 11: Emitter config
   RUNG wire#powerrail
      Contact( #t_Enable )
      wire#w1
      Contact( "DB_Machine".Run )
      Contact( "DB_Machine".AutoCmd.Emit )
      wire#w2
      Coil( "Q_Emit" )
   END_RUNG
   RUNG wire#w1
      Contact( "DB_Machine".ManualMode )
      Contact( "DB_Machine".ManCmd.Emit )
   END_RUNG wire#w2
   // the same network as SCL:
   "Q_Emit" := #t_Enable AND (("DB_Machine".Run AND "DB_Machine".AutoCmd.Emit) OR ("DB_Machine".ManualMode AND "DB_Machine".ManCmd.Emit));
END_REGION

REGION Network 12: Green indicator
   RUNG wire#powerrail
      Contact( "DB_Machine".Run )
      Coil( "Q_GreenIndicator" )
   END_RUNG
   // the same network as SCL:
   "Q_GreenIndicator" := "DB_Machine".Run;
END_REGION

REGION Network 13: Start light
   RUNG wire#powerrail
      Contact( "DB_Machine".Run )
      Coil( "Q_StartLight" )
   END_RUNG
   // the same network as SCL:
   "Q_StartLight" := "DB_Machine".Run;
END_REGION

REGION Network 14: Red indicator
   RUNG wire#powerrail
      I_Contact( "DB_Machine".Run )
      Coil( "Q_RedIndicator" )
   END_RUNG
   // the same network as SCL:
   "Q_RedIndicator" := NOT "DB_Machine".Run;
END_REGION

REGION Network 15: Stop light
   RUNG wire#powerrail
      I_Contact( "DB_Machine".Run )
      Coil( "Q_StopLight" )
   END_RUNG
   // the same network as SCL:
   "Q_StopLight" := NOT "DB_Machine".Run;
END_REGION

REGION Network 16: Yellow indicator
   RUNG wire#powerrail
      Contact( "DB_Machine".Fault )
      wire#w1
      Coil( "Q_YellowIndicator" )
   END_RUNG
   RUNG wire#powerrail
      Contact( "DB_Machine".ManualMode )
   END_RUNG wire#w1
   // the same network as SCL:
   "Q_YellowIndicator" := "DB_Machine".Fault OR "DB_Machine".ManualMode;
END_REGION

REGION Network 17: Reset light
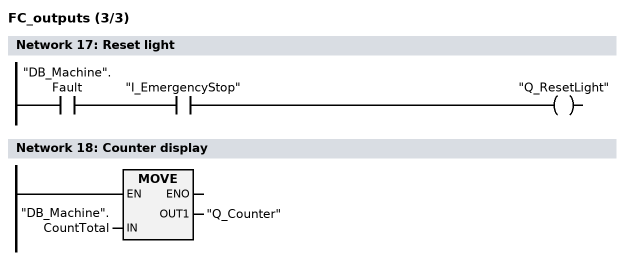
   RUNG wire#powerrail
      Contact( "DB_Machine".Fault )
      Contact( "I_EmergencyStop" )
      Coil( "Q_ResetLight" )
   END_RUNG
   // the same network as SCL:
   "Q_ResetLight" := "DB_Machine".Fault AND "I_EmergencyStop";
END_REGION

REGION Network 18: Counter display
   RUNG wire#powerrail
      Move(in := "DB_Machine".CountTotal, out1 => "Q_Counter")
   END_RUNG
   // the same network as SCL:
   "Q_Counter" := "DB_Machine".CountTotal;
END_REGION
END_FUNCTION

FUNCTION "MHJ-PLC-Lab-Function-S71200" : Void   // FC9000, SCL
{ S7_Optimized_Access := 'TRUE' }
AUTHOR : HoraEmbedded
VERSION : 0.1
   VAR_TEMP
      rdTimeReturn : Int;
      outputTime : DTL;
      SyncVal : Byte;
      forVal : Int;
      forVal_2 : Int;
      Value : Byte;
   END_VAR
   VAR CONSTANT
      CompVal : Byte := 16#34;
      Value_01 : Byte := 16#11;
      Value_01_DW : DWord := 16#A165_D992;
      Value_02_DW : DWord := 16#58BE_4401;
   END_VAR
BEGIN

   #Value:=PEEK(area := 16#82,
        dbNumber := 0,
        byteOffset := 511);
   #Value := #Value + 1;

   POKE(area := 16#82,
        dbNumber := 0,
        byteOffset := 511,
        value := #Value);

   POKE(area:=16#81,
        dbNumber:=0,
        byteOffset:=1016,
        value:=#Value_01_DW);
   POKE(area := 16#81,
        dbNumber := 0,
        byteOffset := 1020,
        value := #Value_02_DW);

   POKE(area := 16#81,
        dbNumber := 0,
        byteOffset := 511,
        value := B#16#00);

   FOR #forVal := 0 TO 120 DO
       FOR #forVal_2:=0 TO 10 DO
           #rdTimeReturn:=RD_SYS_T(#outputTime);
           #rdTimeReturn := WR_SYS_T(#outputTime);
           #rdTimeReturn := RD_SYS_T(#outputTime);
           #rdTimeReturn := WR_SYS_T(#outputTime);
       END_FOR;
       #SyncVal:= PEEK(area := 16#81,
                      dbNumber := 0,
                      byteOffset := 511);
       IF #SyncVal = #CompVal THEN
          GOTO M_1;
       END_IF;
   END_FOR;
   RETURN;

   M_1:
   POKE(area := 16#81,
        dbNumber := 0,
        byteOffset := 511,
        value := B#16#0);
END_FUNCTION

ORGANIZATION_BLOCK "Main"   // OB1, LAD, ProgramCycle
TITLE = Main Program Cycle Execution
{ S7_Optimized_Access := 'TRUE' }
VERSION : 0.1
// Main cyclic block of the S7-1200 PLC. This block coordinates the execution of the entire digital twin program at every PLC scan cycle. It handles the mode manager block to evaluate safety states, runs the main automatic sorting logic sequence, and executes the centralized output gating block to control the physical actuators of the Factory I/O scene.
   VAR_INPUT
      Initial_Call : Bool;   // Initial call of this OB
      Remanence : Bool;   // =True, if remanent data are available
   END_VAR
BEGIN

REGION Network 1
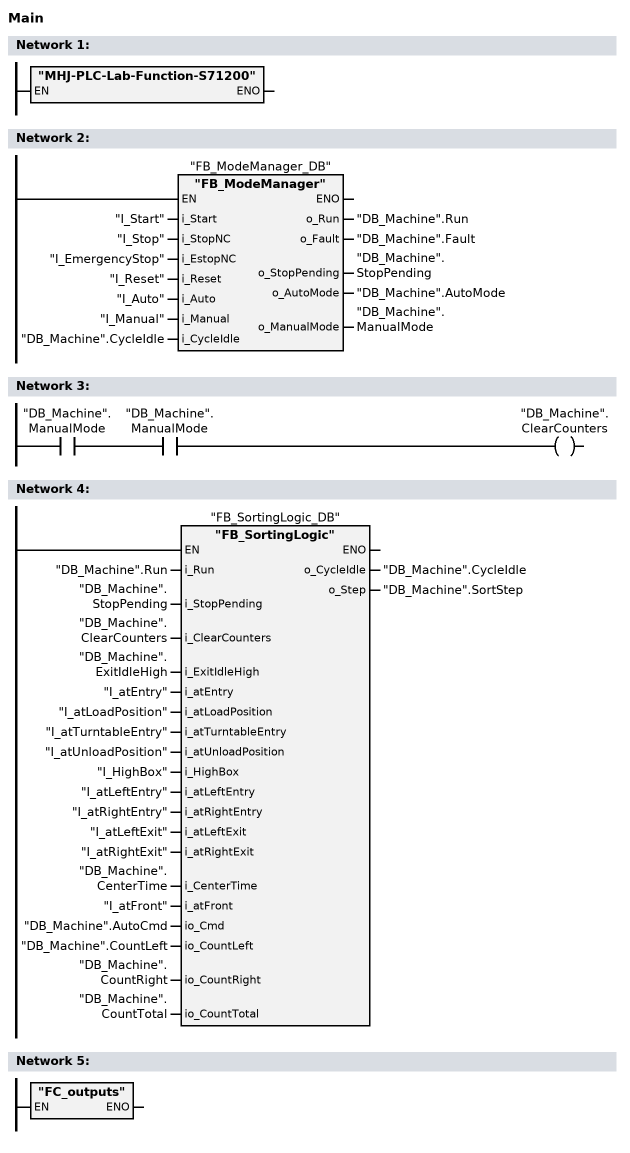
   RUNG wire#powerrail
      "MHJ-PLC-Lab-Function-S71200"()
   END_RUNG
   // the same network as SCL:
   "MHJ-PLC-Lab-Function-S71200"();
END_REGION

REGION Network 2
   RUNG wire#powerrail
      "FB_ModeManager_DB"(i_Start := "I_Start", i_StopNC := "I_Stop", i_EstopNC := "I_EmergencyStop", i_Reset := "I_Reset", i_Auto := "I_Auto", i_Manual := "I_Manual", i_CycleIdle := "DB_Machine".CycleIdle, o_Run => "DB_Machine".Run, o_Fault => "DB_Machine".Fault, o_StopPending => "DB_Machine".StopPending, o_AutoMode => "DB_Machine".AutoMode, o_ManualMode => "DB_Machine".ManualMode)
   END_RUNG
   // the same network as SCL:
   "FB_ModeManager_DB"(i_Start := "I_Start",   // "FB_ModeManager"
                       i_StopNC := "I_Stop",
                       i_EstopNC := "I_EmergencyStop",
                       i_Reset := "I_Reset",
                       i_Auto := "I_Auto",
                       i_Manual := "I_Manual",
                       i_CycleIdle := "DB_Machine".CycleIdle,
                       o_Run => "DB_Machine".Run,
                       o_Fault => "DB_Machine".Fault,
                       o_StopPending => "DB_Machine".StopPending,
                       o_AutoMode => "DB_Machine".AutoMode,
                       o_ManualMode => "DB_Machine".ManualMode);
END_REGION

REGION Network 3
   RUNG wire#powerrail
      Contact( "DB_Machine".ManualMode )
      Contact( "DB_Machine".ManualMode )
      Coil( "DB_Machine".ClearCounters )
   END_RUNG
   // the same network as SCL:
   "DB_Machine".ClearCounters := "DB_Machine".ManualMode AND "DB_Machine".ManualMode;
END_REGION

REGION Network 4
   RUNG wire#powerrail
      "FB_SortingLogic_DB"(i_Run := "DB_Machine".Run, i_StopPending := "DB_Machine".StopPending, i_ClearCounters := "DB_Machine".ClearCounters, i_ExitIdleHigh := "DB_Machine".ExitIdleHigh, i_atEntry := "I_atEntry", i_atLoadPosition := "I_atLoadPosition", i_atTurntableEntry := "I_atTurntableEntry", i_atUnloadPosition := "I_atUnloadPosition", i_HighBox := "I_HighBox", i_atLeftEntry := "I_atLeftEntry", i_atRightEntry := "I_atRightEntry", i_atLeftExit := "I_atLeftExit", i_atRightExit := "I_atRightExit", i_CenterTime := "DB_Machine".CenterTime, i_atFront := "I_atFront", io_Cmd := "DB_Machine".AutoCmd, io_CountLeft := "DB_Machine".CountLeft, io_CountRight := "DB_Machine".CountRight, io_CountTotal := "DB_Machine".CountTotal, o_CycleIdle => "DB_Machine".CycleIdle, o_Step => "DB_Machine".SortStep)
   END_RUNG
   // the same network as SCL:
   "FB_SortingLogic_DB"(i_Run := "DB_Machine".Run,   // "FB_SortingLogic"
                        i_StopPending := "DB_Machine".StopPending,
                        i_ClearCounters := "DB_Machine".ClearCounters,
                        i_ExitIdleHigh := "DB_Machine".ExitIdleHigh,
                        i_atEntry := "I_atEntry",
                        i_atLoadPosition := "I_atLoadPosition",
                        i_atTurntableEntry := "I_atTurntableEntry",
                        i_atUnloadPosition := "I_atUnloadPosition",
                        i_HighBox := "I_HighBox",
                        i_atLeftEntry := "I_atLeftEntry",
                        i_atRightEntry := "I_atRightEntry",
                        i_atLeftExit := "I_atLeftExit",
                        i_atRightExit := "I_atRightExit",
                        i_CenterTime := "DB_Machine".CenterTime,
                        i_atFront := "I_atFront",
                        io_Cmd := "DB_Machine".AutoCmd,
                        io_CountLeft := "DB_Machine".CountLeft,
                        io_CountRight := "DB_Machine".CountRight,
                        io_CountTotal := "DB_Machine".CountTotal,
                        o_CycleIdle => "DB_Machine".CycleIdle,
                        o_Step => "DB_Machine".SortStep);
END_REGION

REGION Network 5
   RUNG wire#powerrail
      "FC_outputs"()
   END_RUNG
   // the same network as SCL:
   "FC_outputs"();
END_REGION
END_ORGANIZATION_BLOCK